% RSLogix 500 project Sensor-Calibration.RSS, saved by version 8.40.00.08 %
PROJECT "UNTITLED"    % processor: Bul.1763 MicroLogix 1100 Series B %

PROGRAM FILES
  LAD 2   16 rungs

DATA FILES
  O0 OUTPUT  4 elements
  I1 INPUT  6 elements
  S2 STATUS  66 elements
  B3 BINARY  1 elements
  T4 TIMER  2 elements
  C5 COUNTER  1 elements
  R6 CONTROL  1 elements
  N7 INTEGER  11 elements
  F8 FLOAT  1 elements

LADDER 2
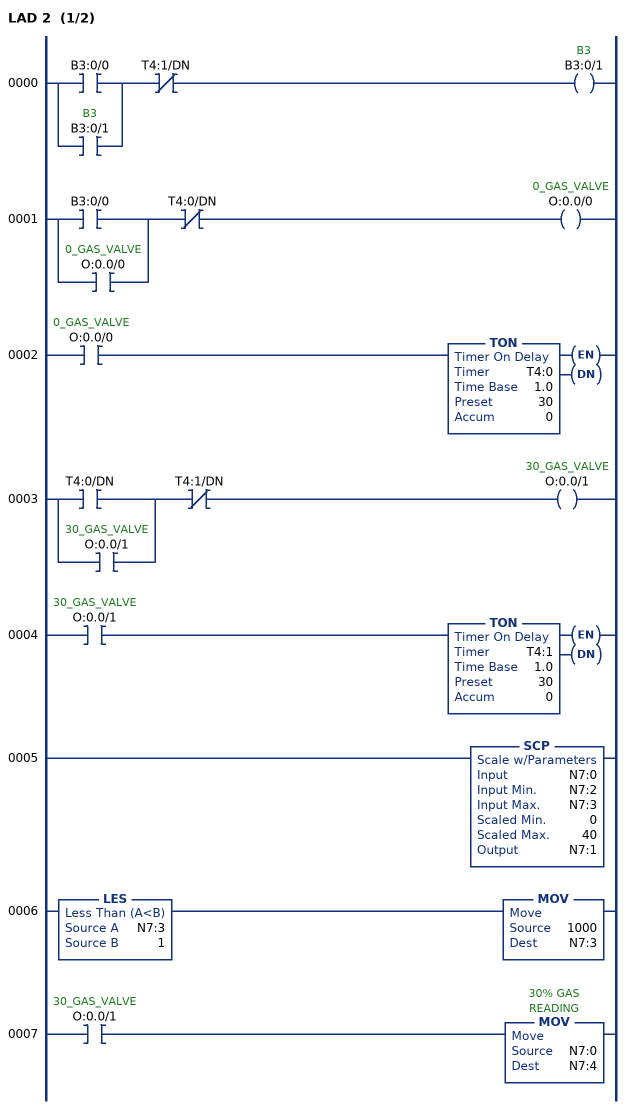
% Rung: 0 %
SOR BST XIC B3:0/0 NXB XIC B3:0/1 BND XIO T4:1/DN OTE B3:0/1 EOR
%   B3:0/1  B3 %
% Rung: 1 %
SOR BST XIC B3:0/0 NXB XIC O:0.0/0 BND XIO T4:0/DN OTE O:0.0/0 EOR
%   O:0.0/0  0_GAS_VALVE %
% Rung: 2 %
SOR XIC O:0.0/0 TON T4:0 1.0 30 0 EOR
%   O:0.0/0  0_GAS_VALVE %
% Rung: 3 %
SOR BST XIC T4:0/DN NXB XIC O:0.0/1 BND XIO T4:1/DN OTE O:0.0/1 EOR
%   O:0.0/1  30_GAS_VALVE %
% Rung: 4 %
SOR XIC O:0.0/1 TON T4:1 1.0 30 0 EOR
%   O:0.0/1  30_GAS_VALVE %
% Rung: 5 %
SOR SCP N7:0 N7:2 N7:3 0 40 N7:1 EOR
% Rung: 6 %
SOR LES N7:3 1 MOV 1000 N7:3 EOR
% Rung: 7 %
SOR XIC O:0.0/1 MOV N7:0 N7:4 EOR
%   O:0.0/1  30_GAS_VALVE %
%   N7:4  "30% GAS READING" %

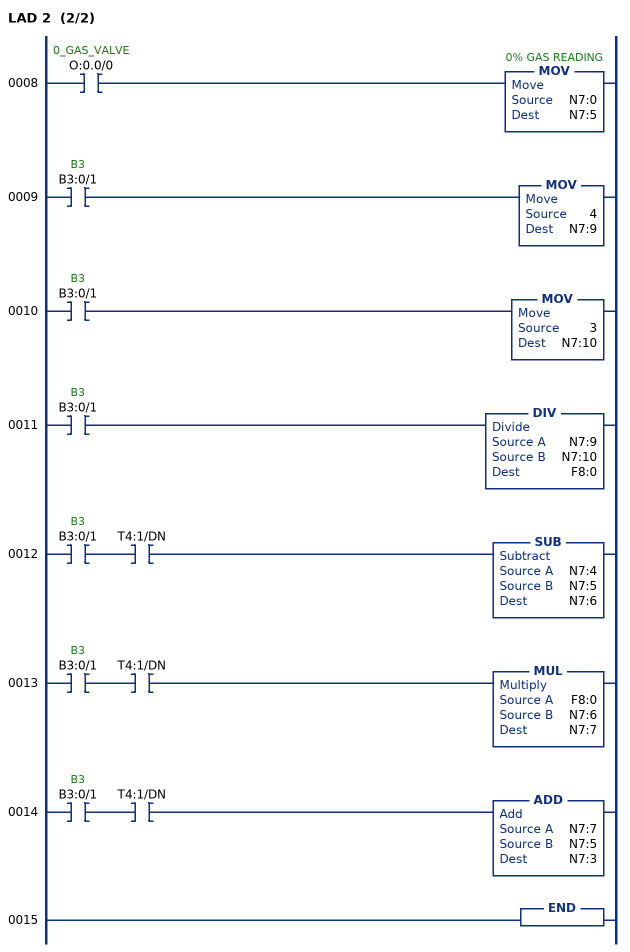
% Rung: 8 %
SOR XIC O:0.0/0 MOV N7:0 N7:5 EOR
%   O:0.0/0  0_GAS_VALVE %
%   N7:5  "0% GAS READING" %
% Rung: 9 %
SOR XIC B3:0/1 MOV 4 N7:9 EOR
%   B3:0/1  B3 %
% Rung: 10 %
SOR XIC B3:0/1 MOV 3 N7:10 EOR
%   B3:0/1  B3 %
% Rung: 11 %
SOR XIC B3:0/1 DIV N7:9 N7:10 F8:0 EOR
%   B3:0/1  B3 %
% Rung: 12 %
SOR XIC B3:0/1 XIC T4:1/DN SUB N7:4 N7:5 N7:6 EOR
%   B3:0/1  B3 %
%   N7:4  "30% GAS READING" %
%   N7:5  "0% GAS READING" %
% Rung: 13 %
SOR XIC B3:0/1 XIC T4:1/DN MUL F8:0 N7:6 N7:7 EOR
%   B3:0/1  B3 %
% Rung: 14 %
SOR XIC B3:0/1 XIC T4:1/DN ADD N7:7 N7:5 N7:3 EOR
%   B3:0/1  B3 %
%   N7:5  "0% GAS READING" %
% Rung: 15 %
SOR END EOR

DATA TABLE (non-zero values as saved)
DATA B3
% B3:0 % 0X0002
DATA T4
% .PRE .ACC %
% T4:0 % 30 0
% T4:1 % 30 0
DATA N7
% N7:0 % 0 0 0 0 0 0 0 0 1 4
% N7:10 % 3
